(* Logix 5000 project; controller Uidaho_Factory vendor 1 type 14 code 165 rev 38.11; software revision 38.00; part 2 of 3 *)
(* tags used below, declared in another part *)
   ESTOP : BOOL;
   GripperTimers : TIMER[10];
   MPO_Auto : BOOL;
   MPO_Compressor_Button : BOOL;
   MPO_Conveyor_Button : BOOL;
   MPO_Feeder_Extend_Button : BOOL;
   MPO_Feeder_Retract_Button : BOOL;
   MPO_Gripper_Lower_Button : BOOL;
   MPO_Gripper_Start : BOOL;
   MPO_Gripper_Toward_Oven_Button : BOOL;
   MPO_Gripper_Toward_Table_Button : BOOL;
   MPO_Gripper_Valve_Button : BOOL;
   MPO_Homing : BOOL;
   MPO_Oven_Door_Button : BOOL;
   MPO_Oven_Light_Button : BOOL;
   MPO_Oven_Start : BOOL;
   MPO_Saw_Button : BOOL;
   MPO_Turntable_CCW_Button : BOOL;
   MPO_Turntable_CW_Button : BOOL;
   MPO_Turntable_Pusher_Button : BOOL;
   MPO_Turntable_Start : BOOL;
   OvenTimers : TIMER[10];
   Step : DINT[20];
   PWM_Outputs : PWM_Out[20];
(* MainProgram, continued *)

ROUTINE MainRoutine   (* ladder *)
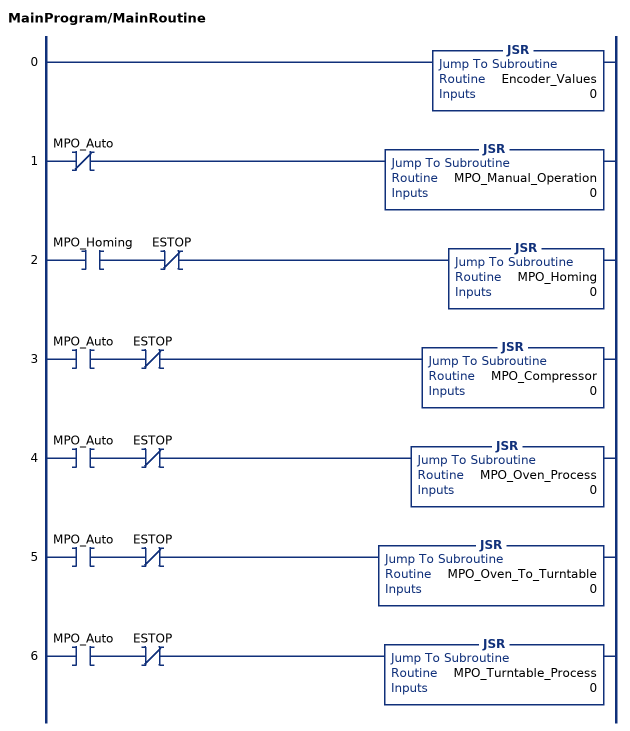
   0: JSR(Encoder_Values,0);
   1: XIO(MPO_Auto)JSR(MPO_Manual_Operation,0);
   2: XIC(MPO_Homing)XIO(ESTOP)JSR(MPO_Homing,0);
   3: XIC(MPO_Auto)XIO(ESTOP)JSR(MPO_Compressor,0);
   4: XIC(MPO_Auto)XIO(ESTOP)JSR(MPO_Oven_Process,0);
   5: XIC(MPO_Auto)XIO(ESTOP)JSR(MPO_Oven_To_Turntable,0);
   6: XIC(MPO_Auto)XIO(ESTOP)JSR(MPO_Turntable_Process,0);
END_ROUTINE

ROUTINE MPO_Compressor   (* ladder *)
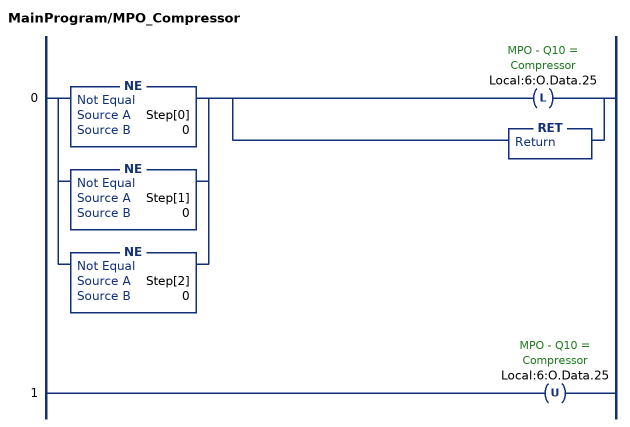
   0: [NE(Step[0],0) ,[NE(Step[1],0) ,NE(Step[2],0) ] ][OTL(Local:6:O.Data.25) ,RET() ];
   1: OTU(Local:6:O.Data.25);
END_ROUTINE

ROUTINE MPO_Homing   (* ladder *)
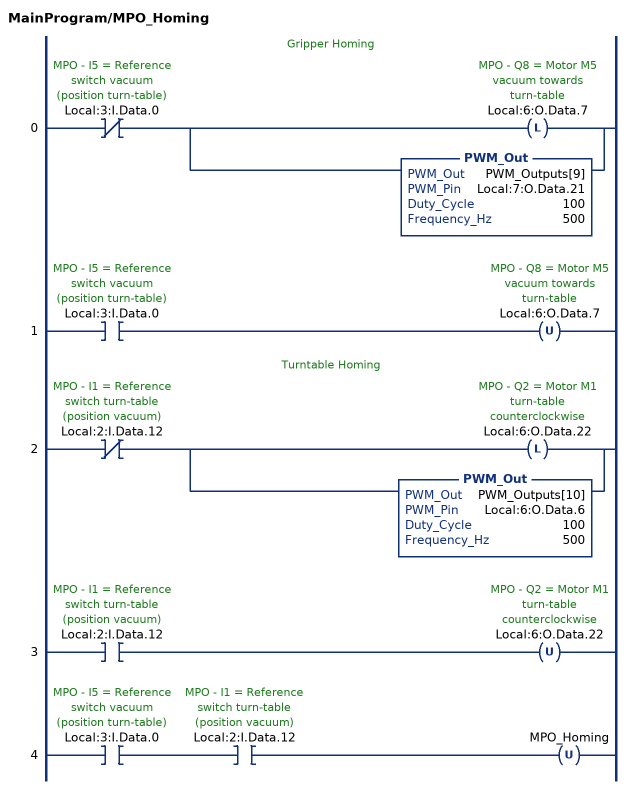
   // Gripper Homing
   0: XIO(Local:3:I.Data.0)[OTL(Local:6:O.Data.7) ,PWM_Out(PWM_Outputs[9],Local:7:O.Data.21,100,500) ];
   1: XIC(Local:3:I.Data.0)OTU(Local:6:O.Data.7);
   // Turntable Homing
   2: XIO(Local:2:I.Data.12)[OTL(Local:6:O.Data.22) ,PWM_Out(PWM_Outputs[10],Local:6:O.Data.6,100,500) ];
   3: XIC(Local:2:I.Data.12)OTU(Local:6:O.Data.22);
   4: XIC(Local:3:I.Data.0)XIC(Local:2:I.Data.12)OTU(MPO_Homing);
END_ROUTINE

ROUTINE MPO_Manual_Operation   (* ladder *)
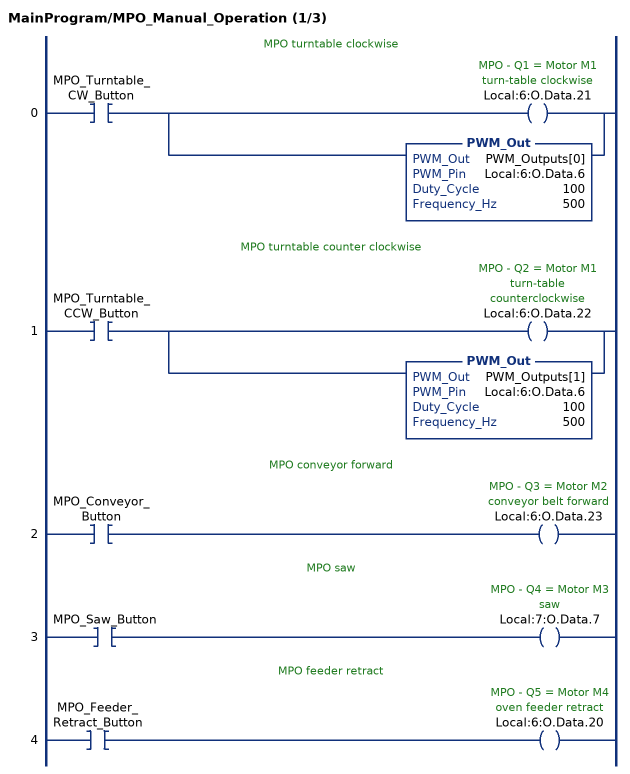
   // MPO turntable clockwise
   0: XIC(MPO_Turntable_CW_Button)[OTE(Local:6:O.Data.21) ,PWM_Out(PWM_Outputs[0],Local:6:O.Data.6,100,500) ];
   // MPO turntable counter clockwise
   1: XIC(MPO_Turntable_CCW_Button)[OTE(Local:6:O.Data.22) ,PWM_Out(PWM_Outputs[1],Local:6:O.Data.6,100,500) ];
   // MPO conveyor forward
   2: XIC(MPO_Conveyor_Button)OTE(Local:6:O.Data.23);
   // MPO saw
   3: XIC(MPO_Saw_Button)OTE(Local:7:O.Data.7);
   // MPO feeder retract
   4: XIC(MPO_Feeder_Retract_Button)OTE(Local:6:O.Data.20);
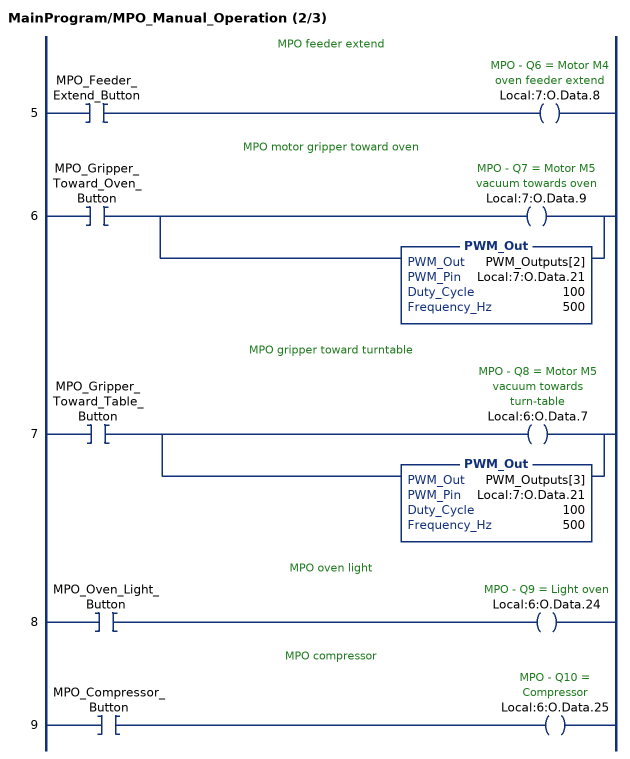
   // MPO feeder extend
   5: XIC(MPO_Feeder_Extend_Button)OTE(Local:7:O.Data.8);
   // MPO motor gripper toward oven
   6: XIC(MPO_Gripper_Toward_Oven_Button)[OTE(Local:7:O.Data.9) ,PWM_Out(PWM_Outputs[2],Local:7:O.Data.21,100,500) ];
   // MPO gripper toward turntable
   7: XIC(MPO_Gripper_Toward_Table_Button)[OTE(Local:6:O.Data.7) ,PWM_Out(PWM_Outputs[3],Local:7:O.Data.21,100,500) ];
   // MPO oven light
   8: XIC(MPO_Oven_Light_Button)OTE(Local:6:O.Data.24);
   // MPO compressor
   9: XIC(MPO_Compressor_Button)OTE(Local:6:O.Data.25);
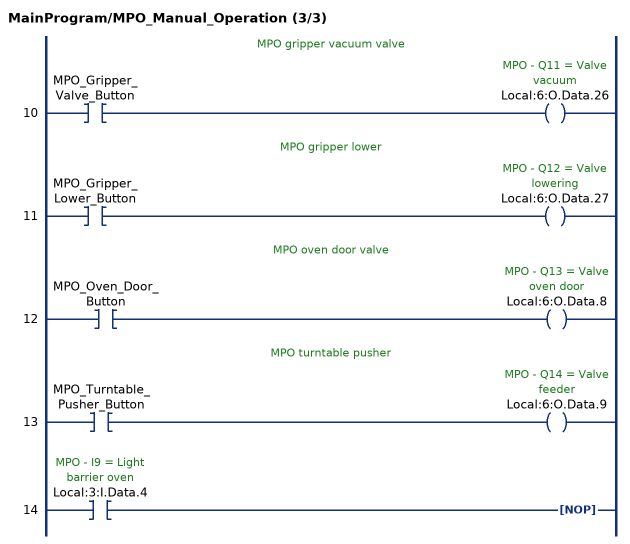
   // MPO gripper vacuum valve
   10: XIC(MPO_Gripper_Valve_Button)OTE(Local:6:O.Data.26);
   // MPO gripper lower
   11: XIC(MPO_Gripper_Lower_Button)OTE(Local:6:O.Data.27);
   // MPO oven door valve
   12: XIC(MPO_Oven_Door_Button)OTE(Local:6:O.Data.8);
   // MPO turntable pusher
   13: XIC(MPO_Turntable_Pusher_Button)OTE(Local:6:O.Data.9);
   14: XIC(Local:3:I.Data.4)NOP();
END_ROUTINE

ROUTINE MPO_Oven_Process   (* ladder *)
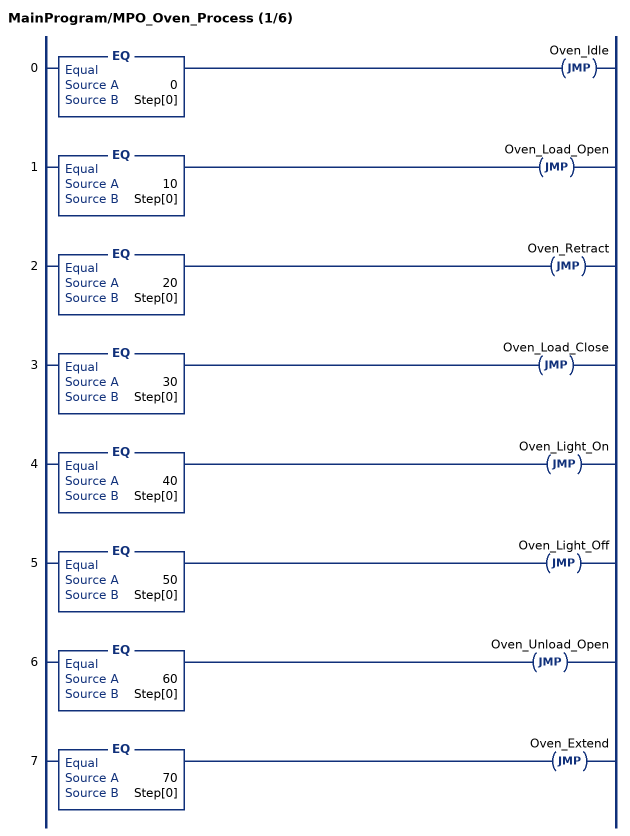
   0: EQ(0,Step[0])JMP(Oven_Idle);
   1: EQ(10,Step[0])JMP(Oven_Load_Open);
   2: EQ(20,Step[0])JMP(Oven_Retract);
   3: EQ(30,Step[0])JMP(Oven_Load_Close);
   4: EQ(40,Step[0])JMP(Oven_Light_On);
   5: EQ(50,Step[0])JMP(Oven_Light_Off);
   6: EQ(60,Step[0])JMP(Oven_Unload_Open);
   7: EQ(70,Step[0])JMP(Oven_Extend);
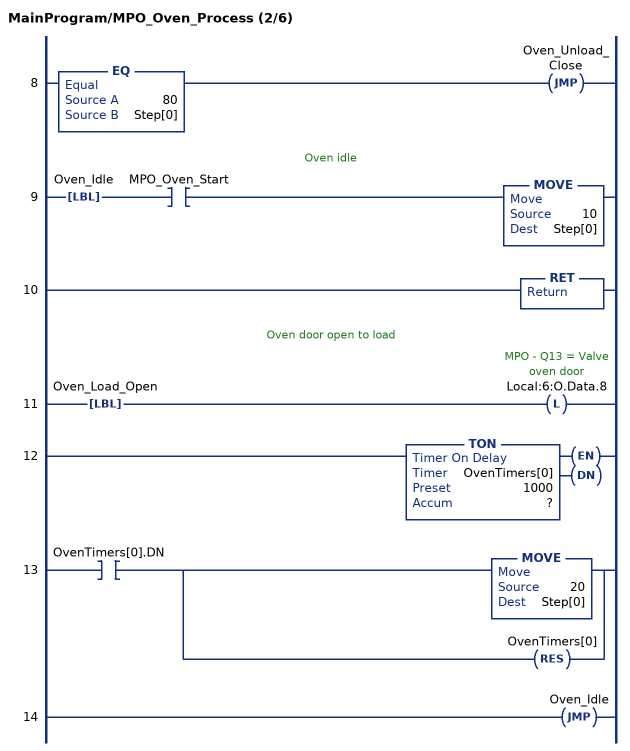
   8: EQ(80,Step[0])JMP(Oven_Unload_Close);
   // Oven idle
   9: LBL(Oven_Idle)XIC(MPO_Oven_Start)MOVE(10,Step[0]);
   10: RET();
   // Oven door open to load
   11: LBL(Oven_Load_Open)OTL(Local:6:O.Data.8);
   12: TON(OvenTimers[0],?,?);
   13: XIC(OvenTimers[0].DN)[MOVE(20,Step[0]) ,RES(OvenTimers[0]) ];
   14: JMP(Oven_Idle);
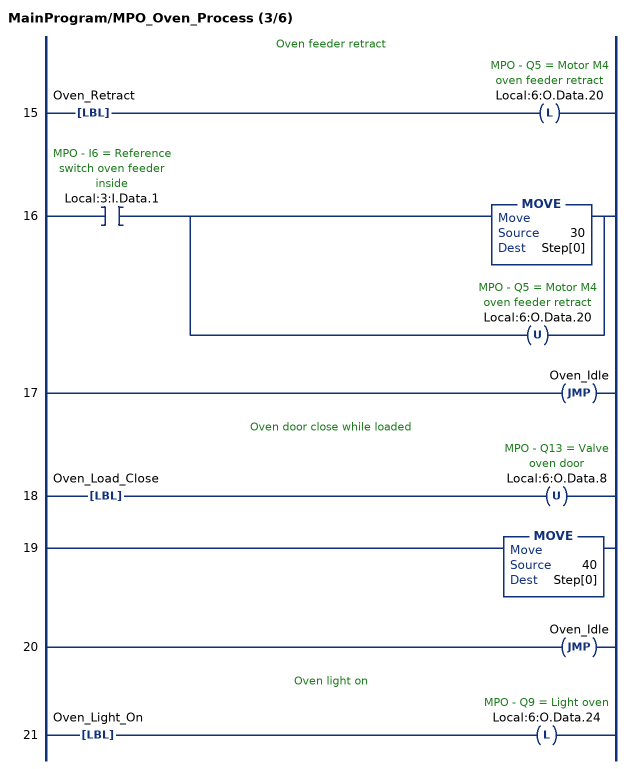
   // Oven feeder retract
   15: LBL(Oven_Retract)OTL(Local:6:O.Data.20);
   16: XIC(Local:3:I.Data.1)[MOVE(30,Step[0]) ,OTU(Local:6:O.Data.20) ];
   17: JMP(Oven_Idle);
   // Oven door close while loaded
   18: LBL(Oven_Load_Close)OTU(Local:6:O.Data.8);
   19: MOVE(40,Step[0]);
   20: JMP(Oven_Idle);
   // Oven light on
   21: LBL(Oven_Light_On)OTL(Local:6:O.Data.24);
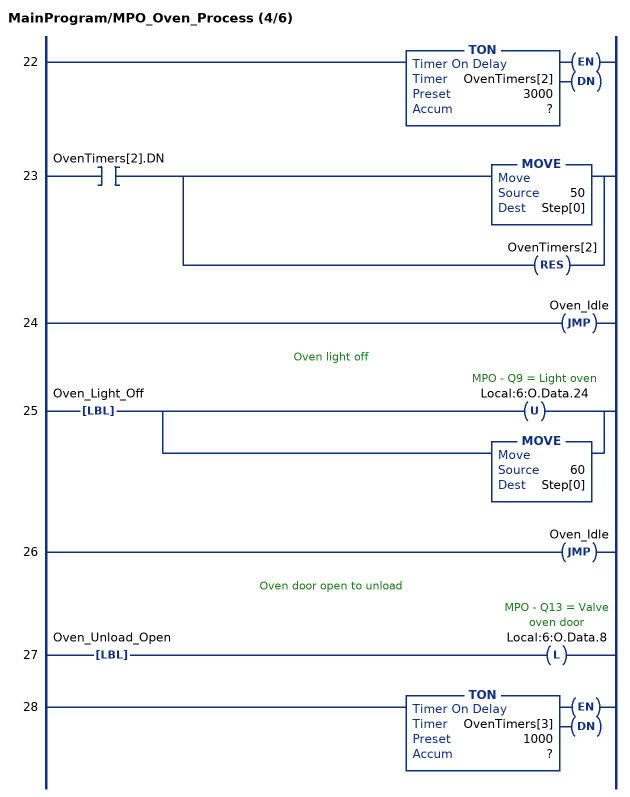
   22: TON(OvenTimers[2],?,?);
   23: XIC(OvenTimers[2].DN)[MOVE(50,Step[0]) ,RES(OvenTimers[2]) ];
   24: JMP(Oven_Idle);
   // Oven light off
   25: LBL(Oven_Light_Off)[OTU(Local:6:O.Data.24) ,MOVE(60,Step[0]) ];
   26: JMP(Oven_Idle);
   // Oven door open to unload
   27: LBL(Oven_Unload_Open)OTL(Local:6:O.Data.8);
   28: TON(OvenTimers[3],?,?);
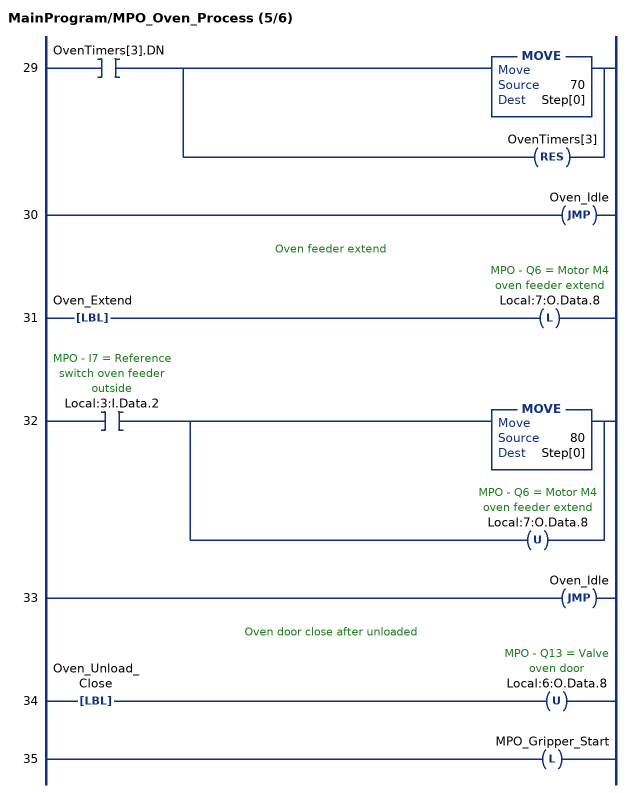
   29: XIC(OvenTimers[3].DN)[MOVE(70,Step[0]) ,RES(OvenTimers[3]) ];
   30: JMP(Oven_Idle);
   // Oven feeder extend
   31: LBL(Oven_Extend)OTL(Local:7:O.Data.8);
   32: XIC(Local:3:I.Data.2)[MOVE(80,Step[0]) ,OTU(Local:7:O.Data.8) ];
   33: JMP(Oven_Idle);
   // Oven door close after unloaded
   34: LBL(Oven_Unload_Close)OTU(Local:6:O.Data.8);
   35: OTL(MPO_Gripper_Start);
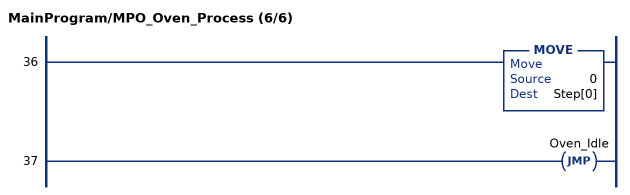
   36: MOVE(0,Step[0]);
   37: JMP(Oven_Idle);
END_ROUTINE

ROUTINE MPO_Oven_To_Turntable   (* ladder *)
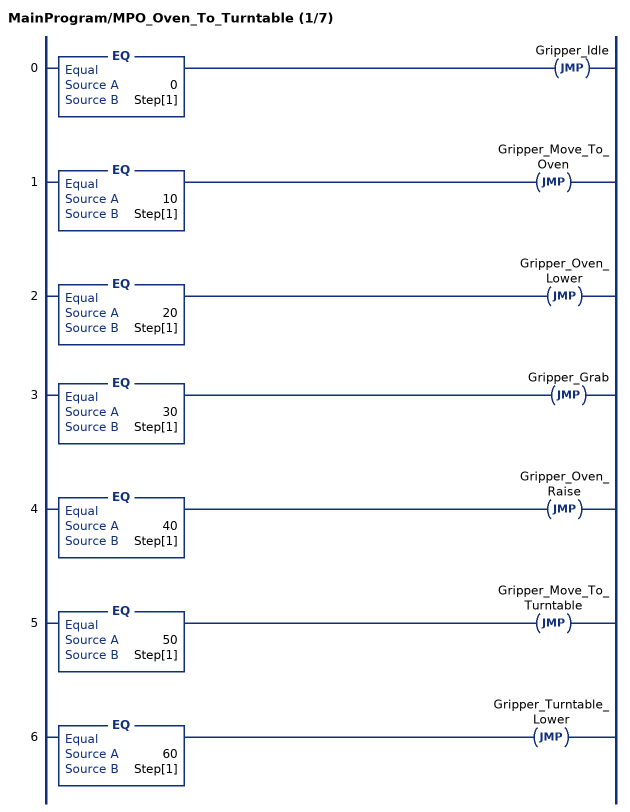
   0: EQ(0,Step[1])JMP(Gripper_Idle);
   1: EQ(10,Step[1])JMP(Gripper_Move_To_Oven);
   2: EQ(20,Step[1])JMP(Gripper_Oven_Lower);
   3: EQ(30,Step[1])JMP(Gripper_Grab);
   4: EQ(40,Step[1])JMP(Gripper_Oven_Raise);
   5: EQ(50,Step[1])JMP(Gripper_Move_To_Turntable);
   6: EQ(60,Step[1])JMP(Gripper_Turntable_Lower);
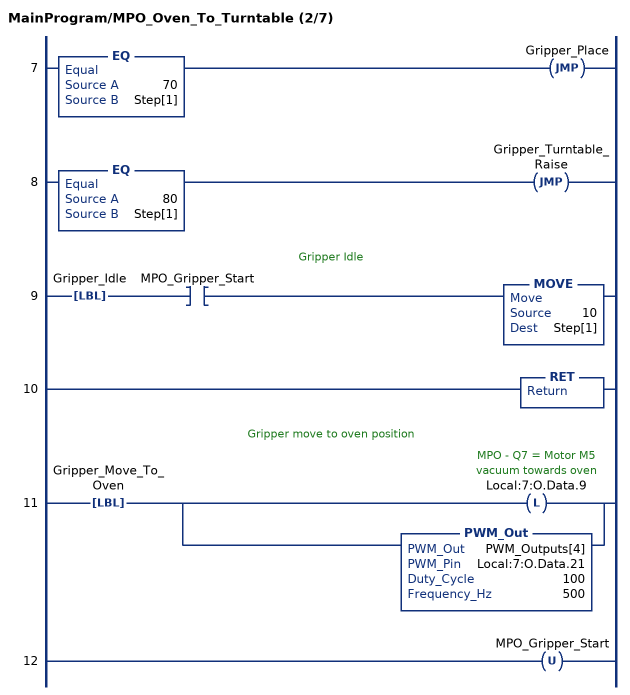
   7: EQ(70,Step[1])JMP(Gripper_Place);
   8: EQ(80,Step[1])JMP(Gripper_Turntable_Raise);
   // Gripper Idle
   9: LBL(Gripper_Idle)XIC(MPO_Gripper_Start)MOVE(10,Step[1]);
   10: RET();
   // Gripper move to oven position
   11: LBL(Gripper_Move_To_Oven)[OTL(Local:7:O.Data.9) ,PWM_Out(PWM_Outputs[4],Local:7:O.Data.21,100,500) ];
   12: OTU(MPO_Gripper_Start);
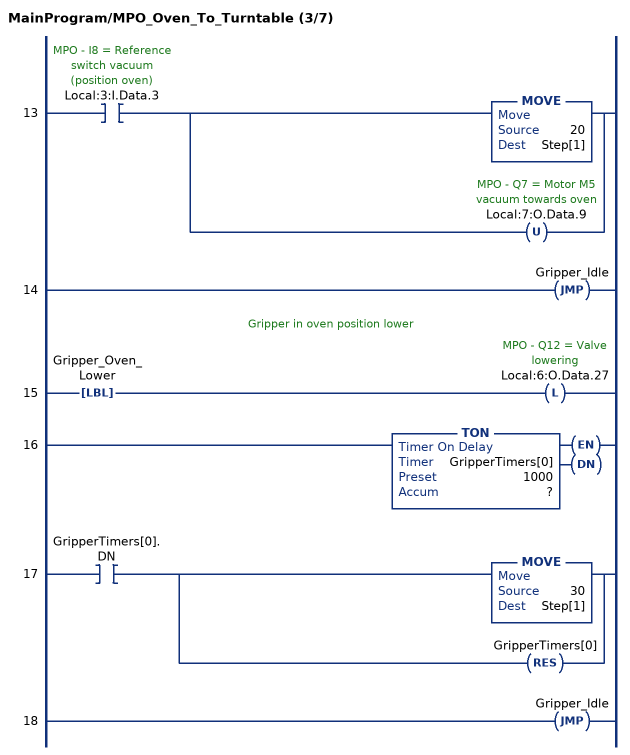
   13: XIC(Local:3:I.Data.3)[MOVE(20,Step[1]) ,OTU(Local:7:O.Data.9) ];
   14: JMP(Gripper_Idle);
   // Gripper in oven position lower
   15: LBL(Gripper_Oven_Lower)OTL(Local:6:O.Data.27);
   16: TON(GripperTimers[0],?,?);
   17: XIC(GripperTimers[0].DN)[MOVE(30,Step[1]) ,RES(GripperTimers[0]) ];
   18: JMP(Gripper_Idle);
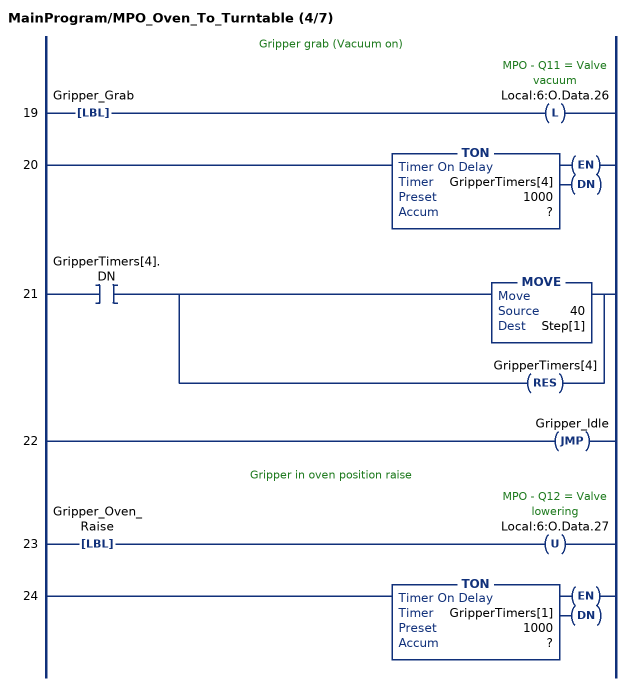
   // Gripper grab (Vacuum on)
   19: LBL(Gripper_Grab)OTL(Local:6:O.Data.26);
   20: TON(GripperTimers[4],?,?);
   21: XIC(GripperTimers[4].DN)[MOVE(40,Step[1]) ,RES(GripperTimers[4]) ];
   22: JMP(Gripper_Idle);
   // Gripper in oven position raise
   23: LBL(Gripper_Oven_Raise)OTU(Local:6:O.Data.27);
   24: TON(GripperTimers[1],?,?);
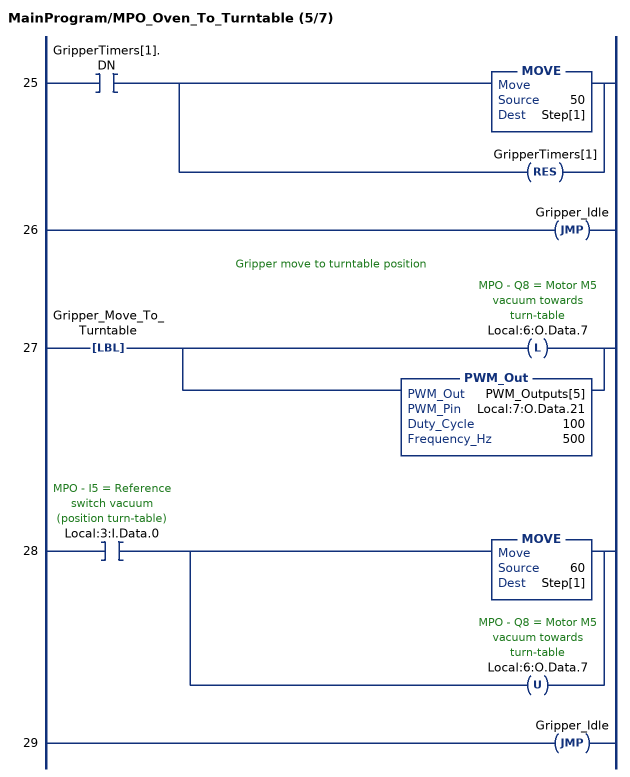
   25: XIC(GripperTimers[1].DN)[MOVE(50,Step[1]) ,RES(GripperTimers[1]) ];
   26: JMP(Gripper_Idle);
   // Gripper move to turntable position
   27: LBL(Gripper_Move_To_Turntable)[OTL(Local:6:O.Data.7) ,PWM_Out(PWM_Outputs[5],Local:7:O.Data.21,100,500) ];
   28: XIC(Local:3:I.Data.0)[MOVE(60,Step[1]) ,OTU(Local:6:O.Data.7) ];
   29: JMP(Gripper_Idle);
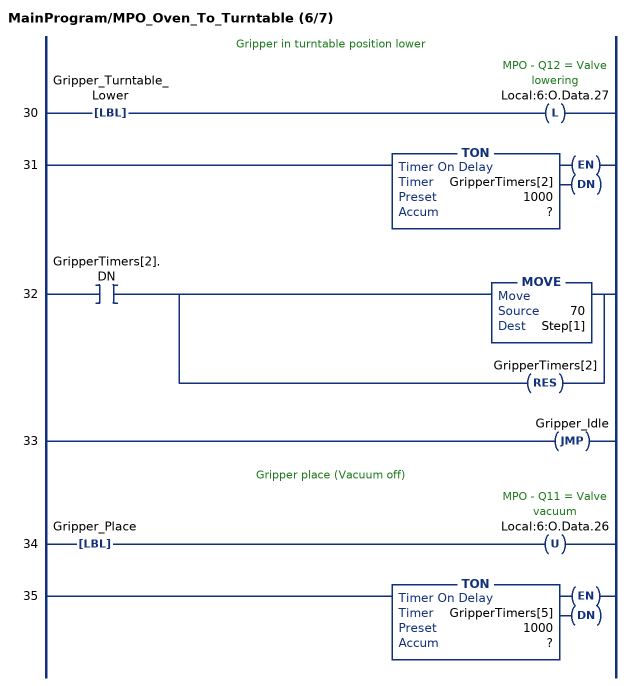
   // Gripper in turntable position lower
   30: LBL(Gripper_Turntable_Lower)OTL(Local:6:O.Data.27);
   31: TON(GripperTimers[2],?,?);
   32: XIC(GripperTimers[2].DN)[MOVE(70,Step[1]) ,RES(GripperTimers[2]) ];
   33: JMP(Gripper_Idle);
   // Gripper place (Vacuum off)
   34: LBL(Gripper_Place)OTU(Local:6:O.Data.26);
   35: TON(GripperTimers[5],?,?);
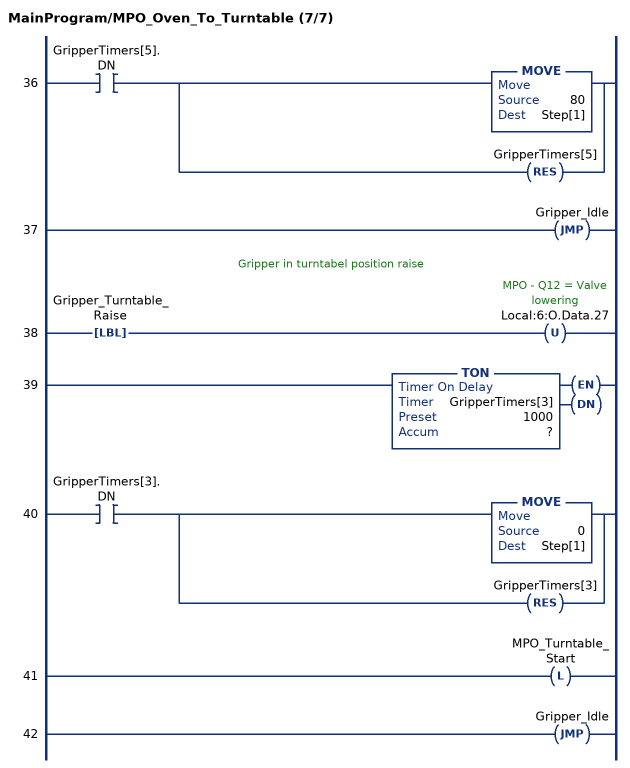
   36: XIC(GripperTimers[5].DN)[MOVE(80,Step[1]) ,RES(GripperTimers[5]) ];
   37: JMP(Gripper_Idle);
   // Gripper in turntabel position raise
   38: LBL(Gripper_Turntable_Raise)OTU(Local:6:O.Data.27);
   39: TON(GripperTimers[3],?,?);
   40: XIC(GripperTimers[3].DN)[MOVE(0,Step[1]) ,RES(GripperTimers[3]) ];
   41: OTL(MPO_Turntable_Start);
   42: JMP(Gripper_Idle);
END_ROUTINE
